{attribute 'qualified_only'}
{attribute 'strict'}
TYPE TestMachineEvents :
(
	Start,
	Stop,
	Abort,
	Reset,
	Clear
);
END_TYPE

(* stored: Version 1.1.0.1, ProductVersion 3.1.4024.12
   DUT TestMachineEvents: Id {9696dd3d-2d8f-08a5-2203-a4d64826f1c2} *)
